TYPE ST_Sample :
STRUCT
    t : LREAL;
    v : LREAL;
END_STRUCT
END_TYPE

(* stored: Version 1.1.0.1
   DUT ST_Sample: Id {6c7f18d1-5fa7-4c87-927b-da332acf5e47} *)
